// TIA Portal V17 export
// export: Created 2026-04-13T11:12:52.796231Z, ExportSetting WithDefaults, DisplayName Totally Integrated Automation Portal, DisplayVersion V17 Update 4, DisplayName TIA Portal Openness, DisplayVersion V17 Update 4, DisplayName TIA Portal Version Control Interface, DisplayVersion V17, DisplayName SINAMICS Startdrive Advanced, DisplayVersion V17, DisplayName SINAMICS Startdrive G130, G150, S120, S150, SINAMICS MV, S210, DisplayVersion V17, DisplayName SINAMICS Startdrive G110M, G120, G120C, G120D, G120P, G115D, DisplayVersion V17, DisplayName STEP 7 Professional, DisplayVersion V17 Update 4, DisplayName STEP 7 Safety, DisplayVersion V17, DisplayName WinCC Professional, DisplayVersion V17 Update 4
TagTable "BY1"
  BY1_MBY等待保压 : Bool  (PLC tag BY1.MBY等待保压, HMI_连接_1, 1 s)
  BY1_MBY正在充气 : Bool  (PLC tag BY1.MBY正在充气, HMI_连接_1, 1 s)
  BY1_MBY保压不佳 : Bool  (PLC tag BY1.MBY保压不佳, HMI_连接_1, 1 s)
  BY1_MBY正在保压 : Bool  (PLC tag BY1.MBY正在保压, HMI_连接_1, 1 s)
  BY1_MBY保压正常 : Bool  (PLC tag BY1.MBY保压正常, HMI_连接_1, 1 s)
  BY1_MBY保压 : Bool  (PLC tag BY1.MBY保压, HMI_连接_1, 1 s)
  BY1_MQT其他阀 : Bool  (PLC tag BY1.MQT其他阀, HMI_连接_1, 1 s)
  BY1_MCQ充气阀 : Bool  (PLC tag BY1.MCQ充气阀, HMI_连接_1, 1 s)
  BY1_当前阶段 : Int  (PLC tag BY1.当前阶段, HMI_连接_1, 1 s)
  BY1_SV低设定 : Real  (PLC tag BY1.SV低设定, HMI_连接_1, 1 s)
  BY1_SV高设定 : Real  (PLC tag BY1.SV高设定, HMI_连接_1, 1 s)
  BY1_SV保压差值 : Real  (PLC tag BY1.SV保压差值, HMI_连接_1, 1 s)
  BY1_SV保压时 : UInt  (PLC tag BY1.SV保压时, HMI_连接_1, 1 s)
  BY1_SV保压分 : UInt  (PLC tag BY1.SV保压分, HMI_连接_1, 1 s)
  BY1_SV保压秒 : UInt  (PLC tag BY1.SV保压秒, HMI_连接_1, 1 s)
  BY1_PV塔内压力 : Real  (PLC tag BY1.PV塔内压力, HMI_连接_1, 1 s)
  BY1_PV保压前 : Real  (PLC tag BY1.PV保压前, HMI_连接_1, 1 s)
  BY1_PV保压后 : Real  (PLC tag BY1.PV保压后, HMI_连接_1, 1 s)
  BY1_PV当前差值 : Real  (PLC tag BY1.PV当前差值, HMI_连接_1, 1 s)
  BY1_PV保压时 : UInt  (PLC tag BY1.PV保压时, HMI_连接_1, 1 s)
  BY1_PV保压分 : UInt  (PLC tag BY1.PV保压分, HMI_连接_1, 1 s)
  BY1_PV保压秒 : UInt  (PLC tag BY1.PV保压秒, HMI_连接_1, 1 s)
  BY1_BY保压重置 : Bool  (PLC tag BY1.BY保压重置, HMI_连接_1, 1 s)
